DATA_BLOCK "DataDb"
{ S7_Optimized_Access := 'TRUE' }
VERSION : 0.1
NON_RETAIN
   VAR
      device { S7_SetPoint := 'False'} : "DeviceData";
   END_VAR


BEGIN

END_DATA_BLOCK

